{attribute 'linkalways'} 
{attribute 'no_explicit_call' := 'This FB is a CLASS and must be accessed using methods or properties'}
{attribute 'enable_dynamic_creation'}
FUNCTION_BLOCK ABSTRACT JsonResponseBuilder IMPLEMENTS I_ResponseBuilder;
VAR
	jsonSaxWriter : FB_JsonSaxWriter;
END_VAR

METHOD PUBLIC AddBase64 : I_ResponseBuilder
VAR_INPUT
	pBytes : POINTER TO BYTE;
	nBytes : DINT;
END_VAR
jsonSaxWriter.AddBase64(pBytes, nBytes);
AddBase64 := THIS^;
END_METHOD

METHOD PUBLIC AddBool : I_ResponseBuilder
VAR_INPUT
	Value : BOOL;
END_VAR
jsonSaxWriter.AddBool(Value);
AddBool := THIS^;
END_METHOD

METHOD PUBLIC AddDateTime : I_ResponseBuilder
VAR_INPUT
	Value : DATE_AND_TIME;
END_VAR
jsonSaxWriter.AddDateTime(Value);
AddDateTime := THIS^;
END_METHOD

METHOD PUBLIC AddDcTime : I_ResponseBuilder
VAR_INPUT
	Value : DCTIME;
END_VAR
jsonSaxWriter.AddDcTime(Value);
AddDcTime := THIS^;
END_METHOD

METHOD PUBLIC AddDint : I_ResponseBuilder
VAR_INPUT
	Value : DINT;
END_VAR
jsonSaxWriter.AddDint(Value);
AddDint := THIS^;
END_METHOD

METHOD PUBLIC AddFileTime : I_ResponseBuilder
VAR_INPUT
	Value : FILETIME;
END_VAR
jsonSaxWriter.AddFileTime(Value);
AddFileTime := THIS^;
END_METHOD

METHOD PUBLIC AddHexBinary : I_ResponseBuilder
VAR_INPUT
	pBytes : POINTER TO BYTE;
	nBytes : DINT;
END_VAR
jsonSaxWriter.AddHexBinary(pBytes, nBytes);
AddHexBinary := THIS^;
END_METHOD

METHOD PUBLIC AddKey : I_ResponseBuilder
VAR_INPUT
	Key : T_MAXSTRING;
END_VAR
jsonSaxWriter.AddKey(Key);
AddKey := THIS^;
END_METHOD

METHOD PUBLIC AddKeyBase64 : I_ResponseBuilder
VAR_INPUT
	Key : T_MAXSTRING;
	pBytes : POINTER TO BYTE;
	nBytes : DINT;
END_VAR
jsonSaxWriter.AddKey(Key);
jsonSaxWriter.AddBase64(pBytes, nBytes);
AddKeyBase64 := THIS^;
END_METHOD

METHOD PUBLIC AddKeyBool : I_ResponseBuilder
VAR_INPUT
	Key : T_MAXSTRING;
	Value : BOOL;
END_VAR
jsonSaxWriter.AddKeyBool(Key,Value);
AddKeyBool := THIS^;
END_METHOD

METHOD PUBLIC AddKeyDateTime : I_ResponseBuilder
VAR_INPUT
	Key : T_MAXSTRING;
	Value : DATE_AND_TIME;
END_VAR
jsonSaxWriter.AddKeyDateTime(Key,Value);
AddKeyDateTime := THIS^;
END_METHOD

METHOD PUBLIC AddKeyDcTime : I_ResponseBuilder
VAR_INPUT
	Key : T_MAXSTRING;
	Value : DCTIME;
END_VAR
jsonSaxWriter.AddKeyDcTime(Key,Value);
AddKeyDcTime := THIS^;
END_METHOD

METHOD PUBLIC AddKeyDint : I_ResponseBuilder
VAR_INPUT
	Key : T_MAXSTRING;
	Value : DINT;
END_VAR
jsonSaxWriter.AddKeyNumber(Key,Value);
AddKeyDint := THIS^;
END_METHOD

METHOD PUBLIC AddKeyFileTime : I_ResponseBuilder
VAR_INPUT
	Key : T_MAXSTRING;
	Value : FILETIME;
END_VAR
jsonSaxWriter.AddKeyFileTime(Key,Value);
AddKeyFileTime := THIS^;
END_METHOD

METHOD PUBLIC AddKeyHexBinary : I_ResponseBuilder
VAR_INPUT
	Key : T_MAXSTRING;
	pBytes : POINTER TO BYTE;
	nBytes : DINT;
END_VAR
jsonSaxWriter.AddKey(Key);
jsonSaxWriter.AddHexBinary(pBytes, nBytes);
AddKeyHexBinary := THIS^;
END_METHOD

METHOD PUBLIC AddKeyLint : I_ResponseBuilder
VAR_INPUT
	Key : T_MAXSTRING;
	Value : LINT;
END_VAR
jsonSaxWriter.AddKey(Key);
jsonSaxWriter.AddLreal(Value);
AddKeyLint := THIS^;
END_METHOD

METHOD PUBLIC AddKeyLreal : I_ResponseBuilder
VAR_INPUT
	Key : T_MAXSTRING;
	Value : LREAL;
END_VAR
jsonSaxWriter.AddKeyLreal(Key,Value);
AddKeyLreal := THIS^;
END_METHOD

METHOD PUBLIC AddKeyNull : I_ResponseBuilder
VAR_INPUT
	Key : T_MAXSTRING;
END_VAR
jsonSaxWriter.AddKeyNull(Key);
AddKeyNull := THIS^;
END_METHOD

METHOD PUBLIC AddKeyReal : I_ResponseBuilder
VAR_INPUT
	Key : T_MAXSTRING;
	Value : REAL;
END_VAR
jsonSaxWriter.AddKey(Key);
jsonSaxWriter.AddReal(Value);
AddKeyReal := THIS^;
END_METHOD

METHOD PUBLIC AddKeyString : I_ResponseBuilder
VAR_INPUT
	Key : T_MAXSTRING;
	Value : T_MAXSTRING;
END_VAR
jsonSaxWriter.AddKeyString(Key,Value);
AddKeyString := THIS^;
END_METHOD

METHOD PUBLIC AddKeyUdint : I_ResponseBuilder
VAR_INPUT
	Key : T_MAXSTRING;
	Value : UDINT;
END_VAR
jsonSaxWriter.AddKey(Key);
jsonSaxWriter.AddUdint(Value);
AddKeyUdint := THIS^;
END_METHOD

METHOD PUBLIC AddKeyUlint : I_ResponseBuilder
VAR_INPUT
	Key : T_MAXSTRING;
	Value : ULINT;
END_VAR
jsonSaxWriter.AddKey(Key);
jsonSaxWriter.AddUlint(Value);
AddKeyUlint := THIS^;
END_METHOD

METHOD PUBLIC AddLint : I_ResponseBuilder
VAR_INPUT
	Value : LINT;
END_VAR
jsonSaxWriter.AddLint(Value);
AddLint := THIS^;
END_METHOD

METHOD PUBLIC AddLreal : I_ResponseBuilder
VAR_INPUT
	Value : LREAL;
END_VAR
jsonSaxWriter.AddLreal(Value);
AddLreal := THIS^;
END_METHOD

METHOD PUBLIC AddNull : I_ResponseBuilder
VAR_INPUT
END_VAR
jsonSaxWriter.AddNull();
AddNull := THIS^;
END_METHOD

METHOD PUBLIC AddReal : I_ResponseBuilder
VAR_INPUT
	Value : REAL;
END_VAR
jsonSaxWriter.AddReal(Value);
AddReal := THIS^;
END_METHOD

METHOD PUBLIC AddString : I_ResponseBuilder
VAR_INPUT
	Value : T_MAXSTRING;
END_VAR
jsonSaxWriter.AddString(Value);
AddString := THIS^;
END_METHOD

METHOD PUBLIC AddUdint : I_ResponseBuilder
VAR_INPUT
	Value : UDINT;
END_VAR
jsonSaxWriter.AddUdint(Value);
AddUdint := THIS^;
END_METHOD

METHOD PUBLIC AddUlint : I_ResponseBuilder
VAR_INPUT
	Value : ULINT;
END_VAR
jsonSaxWriter.AddUlint(Value);
AddUlint := THIS^;
END_METHOD

METHOD PUBLIC EndArray : I_ResponseBuilder
VAR_INPUT
END_VAR
jsonSaxWriter.EndArray();
EndArray := THIS^;
END_METHOD

METHOD PUBLIC EndObject : I_ResponseBuilder
VAR_INPUT
END_VAR
jsonSaxWriter.EndObject();
EndObject := THIS^;
END_METHOD

METHOD PUBLIC ABSTRACT Finalize
VAR_INPUT
END_VAR
END_METHOD

METHOD PUBLIC Reset
VAR_INPUT
END_VAR
jsonSaxWriter.ResetDocument();
END_METHOD

METHOD PUBLIC StartArray : I_ResponseBuilder
VAR_INPUT
END_VAR
jsonSaxWriter.StartArray();
StartArray := THIS^;
END_METHOD

METHOD PUBLIC StartObject : I_ResponseBuilder
VAR_INPUT
END_VAR
jsonSaxWriter.StartObject();
StartObject := THIS^;
END_METHOD

END_FUNCTION_BLOCK

(* stored: Version 1.1.0.1, ProductVersion 3.1.4024.12
   POU JsonResponseBuilder: Id {46cc23c7-d1fb-4fb5-8a1e-bbd7224f0de7}, SpecialFunc None
   Method AddBase64: Id {4b3e748d-ba85-417a-b7ff-fd40641ee2be}
   Method AddBool: Id {8b244953-2331-4c14-b4c2-233f180c4ce7}
   Method AddDateTime: Id {6aca5ea1-1b71-4b05-b884-e40f2cf67420}
   Method AddDcTime: Id {2c3a3a8f-50d1-4f5e-8a3e-00539497354d}
   Method AddDint: Id {fb3bcfb0-fff8-4535-a858-bd0091d4b81b}
   Method AddFileTime: Id {60184c56-6254-4513-b3f3-997cb41909f7}
   Method AddHexBinary: Id {e0b47f84-cf3f-488a-9506-ae3941c2a9a3}
   Method AddKey: Id {24dc1d31-a7a8-4dc3-8da7-f8f5cd3985a2}
   Method AddKeyBase64: Id {c4d939b1-c920-4641-af1d-f65649d7fd9d}
   Method AddKeyBool: Id {00a154c6-524a-4773-9a58-30760eb3d2c0}
   Method AddKeyDateTime: Id {bf2bfd6d-9d27-4c53-9aba-89e8ca075a9c}
   Method AddKeyDcTime: Id {fac6a6f5-4f68-4f56-b2ac-af0f461e69ad}
   Method AddKeyDint: Id {11d73372-5471-4a6a-8228-9565c11f52e7}
   Method AddKeyFileTime: Id {f838397a-d634-4482-858d-33db9270e820}
   Method AddKeyHexBinary: Id {f180dc6f-65b3-4919-8463-568db3df92ac}
   Method AddKeyLint: Id {7510350b-852d-41b5-bdca-f4972876f237}
   Method AddKeyLreal: Id {db5cb8c2-80dd-4ac7-887d-71a29376b468}
   Method AddKeyNull: Id {d4bf33e8-1a26-4e80-901e-836f2b241c70}
   Method AddKeyReal: Id {7634e453-7f61-4154-b659-fc54aca8a5b3}
   Method AddKeyString: Id {ccda3039-b2dc-4653-b178-fc8f42288703}
   Method AddKeyUdint: Id {f9533667-b6a3-45d4-a337-25c097ab37f9}
   Method AddKeyUlint: Id {d789a0dd-877b-4c08-9923-d9a12da62ebb}
   Method AddLint: Id {10b3f128-d63d-4a94-b1aa-25b1f8cf8fb9}
   Method AddLreal: Id {2dff83a0-f1cc-4d83-95a1-fedd5627639b}
   Method AddNull: Id {c3420488-53d6-417e-8c45-bec5a71424ae}
   Method AddReal: Id {3ea261da-db98-448f-a044-3fd5a7f35f4c}
   Method AddString: Id {89d00345-cd84-41ec-aa6f-c9c2159f1ec5}
   Method AddUdint: Id {db681cb1-dddd-4d5d-8cca-7bd9f8dec874}
   Method AddUlint: Id {e1eb61e2-dad9-4232-8345-32512b02b58d}
   Method EndArray: Id {e73f4dd1-792c-48c5-abdf-8804f39eddf6}
   Method EndObject: Id {7e3158a9-6b16-430a-9b41-3fb97e862e95}
   Method Finalize: Id {04ec01a6-4cfb-4172-9918-54074f56a0e9}
   Method Reset: Id {23d5e104-dbce-49af-bb35-899d780a7ae0}
   Method StartArray: Id {b28a9414-dcdf-426b-8e69-52abb1e27053}
   Method StartObject: Id {00981cef-94d7-4475-9700-7e680248306e} *)
